INTERFACE I_NciChannel_GCode EXTENDS I_NciChannelBase

PROPERTY IsMoving : BOOL
GET
END_GET
END_PROPERTY

PROPERTY IsProgramLoaded : BOOL
GET
END_GET
END_PROPERTY

METHOD LoadProgram
VAR_INPUT
	sProgramPath : STRING(255);
END_VAR
END_METHOD

METHOD Start
VAR_INPUT
END_VAR
END_METHOD

END_INTERFACE

(* stored: Version 1.1.0.1, ProductVersion 3.1.4024.15
   Itf I_NciChannel_GCode: Id {7a91496b-baa2-4b9c-9bd6-d47f2d3e317c}
   Property IsMoving: Id {863c3f1d-e3ba-4ca0-b3c8-cdfa03f416b8}
   Get Get: Id {49cc0586-bfa7-4842-a93d-55749afd24ad}
   Property IsProgramLoaded: Id {20083fb0-60e0-44a1-a862-ec7336c142a2}
   Get Get: Id {fd981e8e-6705-4c5f-ae9b-b12f2b0e7e1d}
   Method LoadProgram: Id {20f09308-de81-4286-853c-7c9f23771b69}
   Method Start: Id {e1607d78-d8ee-4b50-8e8d-0575feea8216} *)
